RoboDK station: RoboDK_station.rdk

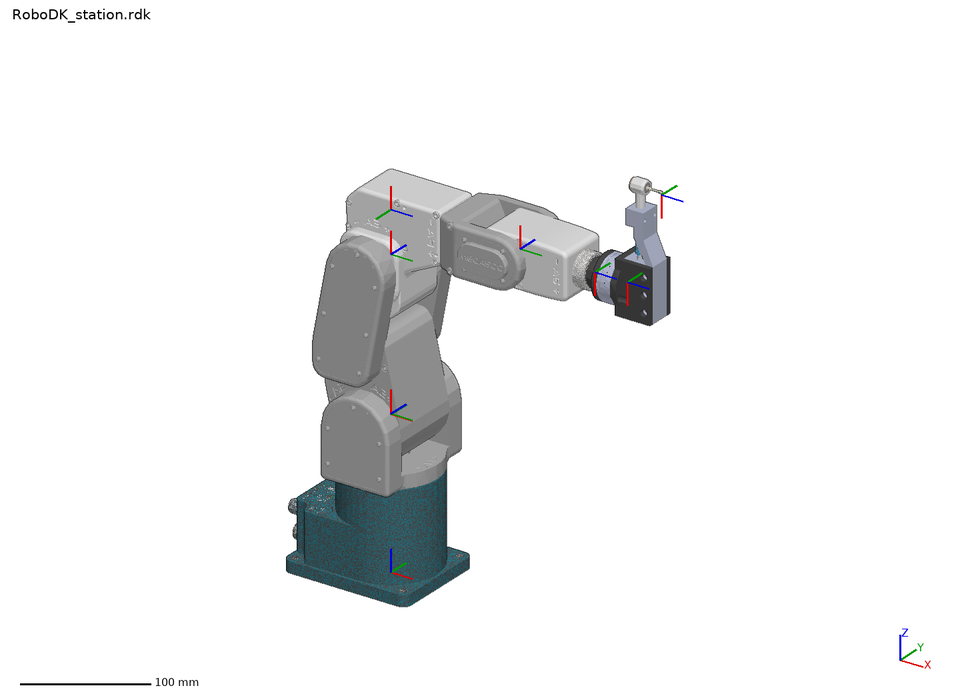
[picture v0: the station drawn from its stored meshes, robots at their saved joint values, targets as dots, program paths as lines]
Station RoboDK_station (saved by RoboDK 5.1.0). Poses are relative to the parent item; angles as X-Y-Z fixed-axis rotations.
  - object main at (0, 0, 0) mm, rotated rx 90 ry 0 rz 90 deg, size 101.4 x 399.3 x 338.5 mm, geometry from main.STEP
  - frame {1} at (0, 0, 44) mm
  - frame {2} at (0, 0, 45) mm, rotated rx 0 ry -90 rz -90 deg
  - frame {3} at (0, 0, 180) mm, rotated rx 0 ry -90 rz -90 deg
  - frame {4} at (0, 0, 218) mm, rotated rx 0 ry -90 rz 180 deg
  - frame {5} at (120, 0, 218) mm, rotated rx 0 ry -90 rz -90 deg
  - frame {6} at (190, 0, 218) mm, rotated rx 0 ry 90 rz 0 deg
  - frame {S} at (220, 0, 218) mm, rotated rx 0 ry 90 rz 0 deg
  - frame {T} at (252, 0, 301) mm, rotated rx 0 ry 90 rz 0 deg
  - frame {0} at (0, 0, -90) mm
